PROGRAM MAIN
VAR	
	HardwareControl : HardwareControl;
END_VAR


HardwareControl();

END_PROGRAM

(* stored: Version 1.1.0.1, ProductVersion 3.1.4024.12
   POU MAIN: Id {58925a0b-bcf4-4828-885e-2cbd0bc812af}, SpecialFunc None *)
